TYPE "UDT_ZC_DISP_TON"
VERSION : 0.1
   STRUCT
      SP : Int := 5;
      ET : Int := 0;
      IN : Bool := false;
      Q : Bool := false;
   END_STRUCT;

END_TYPE

